FUNCTION_BLOCK SOL_MDLL (* Locally-Coupled Solenoid Model *)
  (* Standard: 61499-1; Classification: Model; ApplicationDomain: Simulation; Function: Material Handling; Type: Conveyor *)
  (* Version 0.0, 2004-09-23, JHC, Rockwell Automation, Converted to distributed clock. *)
  (* Compiler header: package fb.rt.mva; import fb.rt.math.*; import fb.rt.net.*; *)
  (* Compiler classdef: public class SOL_MDLL1 extends FBMVCD *)
  (* Compiler Java Sun JDK 1.4.2 *)
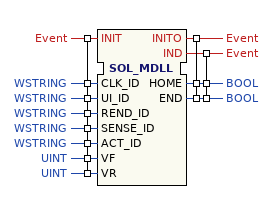
  EVENT_INPUT
    INIT WITH REND_ID, ACT_ID, VF, CLK_ID, UI_ID, VR, SENSE_ID; (* Initialize *)
  END_EVENT
  EVENT_OUTPUT
    INITO WITH END, HOME; (* View Initialized *)
    IND WITH HOME, END; (* Change in Sensor Data *)
  END_EVENT
  VAR_INPUT
    CLK_ID : WSTRING := "SIM_CLK"; (* Simulation clock channel ID *)
    UI_ID : WSTRING; (* User input channel ID from View *)
    REND_ID : WSTRING; (* Rendering data channel ID to View *)
    SENSE_ID : WSTRING; (* Sensor data channel ID to Controller *)
    ACT_ID : WSTRING; (* Actuator data channel ID from Controller *)
    VF : UINT := 50; (* Forward Speed in % per CLK event *)
    VR : UINT := 50; (* Retract Speed in % per CLK event *)
  END_VAR
  VAR_OUTPUT
    HOME : BOOL; (* Solenoid Fully Retracted *)
    END : BOOL; (* Solenoid Fully Advanced *)
  END_VAR
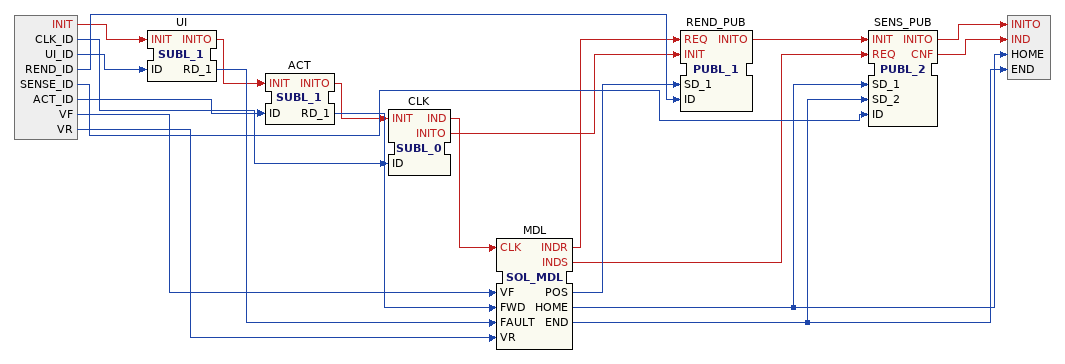
  FBS
    ACT : SUBL_1;
    MDL : SOL_MDL;
    REND_PUB : PUBL_1;
    CLK : SUBL_0;
    UI : SUBL_1;
    SENS_PUB : PUBL_2;
  END_FBS
  EVENT_CONNECTIONS
    MDL.INDR TO REND_PUB.REQ;
    CLK.IND TO MDL.CLK;
    INIT TO UI.INIT;
    UI.INITO TO ACT.INIT;
    ACT.INITO TO CLK.INIT;
    CLK.INITO TO REND_PUB.INIT;
    REND_PUB.INITO TO SENS_PUB.INIT;
    MDL.INDS TO SENS_PUB.REQ;
    SENS_PUB.INITO TO INITO;
    SENS_PUB.CNF TO IND;
  END_CONNECTIONS
  DATA_CONNECTIONS
    MDL.POS TO REND_PUB.SD_1;
    VF TO MDL.VF;
    ACT.RD_1 TO MDL.FWD;
    UI.RD_1 TO MDL.FAULT;
    VR TO MDL.VR;
    CLK_ID TO CLK.ID;
    UI_ID TO UI.ID;
    ACT_ID TO ACT.ID;
    REND_ID TO REND_PUB.ID;
    MDL.HOME TO SENS_PUB.SD_1;
    MDL.END TO SENS_PUB.SD_2;
    SENSE_ID TO SENS_PUB.ID;
    MDL.HOME TO HOME;
    MDL.END TO END;
  END_CONNECTIONS
END_FUNCTION_BLOCK
